{attribute 'qualified_only' := ''}
{attribute 'strict' := ''}
TYPE E_PackageSeparationState :
(
	NORMAL := 0,
	START_SEPARATION := 10,
	CONVEYOR_2_TRACKING := 20,
	CONVEYOR_3_TRACKING := 30,
	FINISH_SEPARATION := 40
);
END_TYPE

(* stored: Version 1.1.0.1
   DUT E_PackageSeparationState: Id {5062d5e8-cb34-4295-8849-9d00c37921d7} *)
